Universal Robots PolyScope program: CircularPath_1.urp

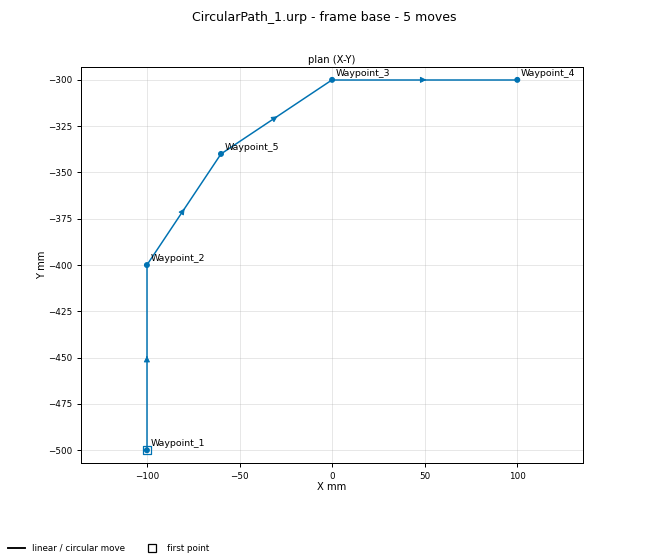
[picture p0: tool path of CircularPath_1.urp in frame base, 5 of 5 moves have a stored position in this frame; points joined in program order, loops and branches not executed]
ProgramRoot directory=/home/ur/ursim-1.5/programs/templates/CircularPathUsingMoveP; kinematics=(a=[0, -0.425, -0.39243, 0, 0, 0], d=[0.0892, 0, 0, 0.109, 0.093, 0.082], alpha=[1.5708, 0, 0, 1.5708, -1.5708, 0], deltaTheta=[0, 0, 0, 0, 0, 0], status=notInitialized); name=CircularPath_1; programVersion=(project__name=PolyScope, major__version=1, minor__version=5, svn__revision=7526, build__date=Dec 21 2011, 13:03:24); robotEnvironmentFileName=default
  MainProgram cartesianAcceleration=1.2; cartesianSpeed=0.25; jointAcceleration=1.3962634015954636; jointSpeed=1.0471975511965976; moveAsFastAsPossible=true; sharedProcessMoveBlendRadius=0.025; featureReference=(installationNameReference=Base); motionType=JOINT_SPACE
    Move cartesianAcceleration=1.2; cartesianSpeed=0.25; jointAcceleration=1.3962634015954636; jointSpeed=1.0471975511965976; moveAsFastAsPossible=true; sharedProcessMoveBlendRadius=0.0020; featureReference=(installationNameReference=Base); motionType=PROCESS_MOVE
      Waypoint blendRadius=0.0; cartesianAcceleration=1.2; cartesianSpeed=0.25; jointAcceleration=1.3962634015954636; jointSpeed=1.0471975511965976; nextMotionTime=2.0; useSharedBlendParameter=true; useSharedParameters=true; position=TCP in base x=-100 y=-500 z=200 mm, rx=0 ry=3.14 rz=0.0006 rad; joints [-88.982, -101.255, -113.55, -55.216, 90.094, 1.018] deg; positionType=FIXED_POSITION; waypointPoseInFeatureCoordinates=(pos=(x=-0.09999999999998957, y=-0.5000000000000082, z=0.1999998668199792), rot=(x=-5.308256505009962E-7, y=3.139954578393098, z=6.183385988155127E-4)); name=Waypoint_1
      Waypoint blendRadius=0.0; cartesianAcceleration=1.2; cartesianSpeed=0.25; jointAcceleration=1.3962634015954636; jointSpeed=1.0471975511965976; nextMotionTime=2.0; useSharedBlendParameter=true; useSharedParameters=true; position=TCP in base x=-100 y=-400 z=200 mm, rx=0 ry=3.14 rz=0.0006 rad; joints [-88.727, -88.409, -127.833, -53.779, 90.094, 1.273] deg; positionType=FIXED_POSITION; waypointPoseInFeatureCoordinates=(pos=(x=-0.09999999999998924, y=-0.40000000000000957, z=0.19999986681998774), rot=(x=-5.308256790783317E-7, y=3.1399545783933682, z=6.183385987292099E-4)); name=Waypoint_2
      CircleMove insertableAsSuppressedNode=true; description=<html>A circle move is made with two waypoints. The first one specifying a via point on the circular arc, and the second one being the endpoint of the movement. The robot will start the circle movement from its current position, and then move through the two specified waypoints. The orientation change of the tool through the circle move is determined only by the starting orientation and the orientation at the endpoint, thus the orientation of the via point does not influence the circle move. <p><p> A CircleMove must always be preceeded by a waypoint under the same MoveP.</html>; name=CircleMove
        Waypoint blendRadius=0.0; cartesianAcceleration=1.2; cartesianSpeed=0.25; jointAcceleration=1.3962634015954636; jointSpeed=1.0471975511965976; nextMotionTime=2.0; useSharedBlendParameter=true; useSharedParameters=true; position=TCP in base x=-60 y=-340 z=200 mm, rx=0 ry=3.14 rz=0.0006 rad; joints [-81.628, -78.006, -136.607, -55.396, 90.096, 8.372] deg; positionType=FIXED_POSITION; waypointPoseInFeatureCoordinates=(pos=(x=-0.05999999798496541, y=-0.3399999959114223, z=0.19999986681999668), rot=(x=-5.308260676994364E-7, y=3.139954579717172, z=6.183382191660831E-4)); name=Waypoint_5
        Waypoint blendRadius=0.0; cartesianAcceleration=1.2; cartesianSpeed=0.25; jointAcceleration=1.3962634015954636; jointSpeed=1.0471975511965976; nextMotionTime=2.0; useSharedBlendParameter=true; useSharedParameters=true; position=TCP in base x=0 y=-300 z=200 mm, rx=0 ry=3.14 rz=0.0006 rad; joints [-68.723, -69.674, -141.948, -58.365, 90.096, 21.277] deg; positionType=FIXED_POSITION; waypointPoseInFeatureCoordinates=(pos=(x=-1.9283241666086012E-14, y=-0.29999999999998705, z=0.19999986682000667), rot=(x=-5.308255817083467E-7, y=3.139954578393368, z=6.183385987560061E-4)); name=Waypoint_3
      Waypoint blendRadius=0.05; cartesianAcceleration=1.2; cartesianSpeed=0.25; jointAcceleration=1.3962634015954636; jointSpeed=1.0471975511965976; nextMotionTime=2.0; stoppoint=true; useSharedBlendParameter=true; useSharedParameters=true; position=TCP in base x=100 y=-300 z=200 mm, rx=0 ry=3.14 rz=0.0006 rad; joints [-51.426, -72.815, -140.108, -57.036, 90.087, 38.574] deg; positionType=FIXED_POSITION; waypointPoseInFeatureCoordinates=(pos=(x=0.09999999999999121, y=-0.2999999999999814, z=0.19999986682001572), rot=(x=-5.308255965683186E-7, y=3.1399545783933682, z=6.183385986190898E-4)); name=Waypoint_4
